TYPE ST_SYSTEM_Door :
STRUCT
	bClearConveyorQueue						: BOOL;
	bClearPackerQueue							: BOOL;
	aClearCaseQueue							: ARRAY[1..cMAX_CASE_QUEUE] OF BOOL;
END_STRUCT
END_TYPE

(* stored: Version 1.1.0.1
   DUT ST_SYSTEM_Door: Id {25e34554-b43e-4e55-b7f2-69a3821f8eeb} *)
